   Chain7Long.Drive.ACT.CMD.HwPosOvertravel_Dis := FALSE;
   Chain7Long.Drive.ACT.CMD.HwNegOvertravel_Dis := FALSE;
   Chain7Long.Drive.ACT.CMD.HwOvertravel_MSG_En := FALSE;
   Chain7Long.Drive.ACT.CMD.OneShootMove := FALSE;
   Chain7Long.Drive.ACT.CMD.Move_Type := 3;
   Chain7Long.Drive.ACT.CMD.Target_Pos := 0.0;
   Chain7Long.Drive.ACT.CMD.Speed := 50.0;
   Chain7Long.Drive.ACT.CMD.Acceleration := 300.0;
   Chain7Long.Drive.ACT.CMD.Deceleration := 300.0;
   Chain7Long.Drive.ACT.CMD.Torque_Limit := 30.0;
   Chain7Long.Drive.ACT.CMD.Gear_Ratio := 0.0;
   Chain7Long.Drive.ACT.CMD.Mccp_Length := 2;
   Chain7Long.Drive.ACT.CMD.Mccp_StartSlope := 0.0;
   Chain7Long.Drive.ACT.CMD.Mccp_EndSlope := 0.0;
   Chain7Long.Drive.ACT.CMD.Mapc_Direction := 1;
   Chain7Long.Drive.ACT.CMD.Mapc_SlaveScaling := 1.0;
   Chain7Long.Drive.ACT.CMD.Mapc_MasterScaling := 1.0;
   Chain7Long.Drive.ACT.CMD.Mapc_MasterLockPosition := 0.0;
   Chain7Long.Drive.ACT.CMD.Mapc_CamLockPosition := 0.0;
   Chain7Long.Drive.ACT.CMD.Cam[0].leadingValueStart := 0.0;
   Chain7Long.Drive.ACT.CMD.Cam[1].leadingValueStart := 162.0;
   Chain7Long.Drive.ACT.CMD.Cam[2..39].leadingValueStart := 0.0;
   Chain7Long.Drive.ACT.CMD.Cam[0].leadingValueEnd := 162.0;
   Chain7Long.Drive.ACT.CMD.Cam[1].leadingValueEnd := 360.0;
   Chain7Long.Drive.ACT.CMD.Cam[2..39].leadingValueEnd := 0.0;
   Chain7Long.Drive.ACT.CMD.Cam[0].followingValueStart := 0.0;
   Chain7Long.Drive.ACT.CMD.Cam[1].followingValueStart := 406.399993896484;
   Chain7Long.Drive.ACT.CMD.Cam[2..39].followingValueStart := 0.0;
   Chain7Long.Drive.ACT.CMD.Cam[0..1].followingValueEnd := 406.399993896484;
   Chain7Long.Drive.ACT.CMD.Cam[2..39].followingValueEnd := 0.0;
   Chain7Long.Drive.ACT.CMD.Cam[0..39].geoVeloStart := 0.0;
   Chain7Long.Drive.ACT.CMD.Cam[0..39].geoVeloEnd := 0.0;
   Chain7Long.Drive.ACT.CMD.Cam[0..39].geoAccelStart := 0.0;
   Chain7Long.Drive.ACT.CMD.Cam[0..39].geoAccelEnd := 0.0;
   Chain7Long.Drive.ACT.CMD.Cam[0..39].geoJerkStart := 0.0;
   Chain7Long.Drive.ACT.CMD.Cam[0..39].geoJerkEnd := 0.0;
   Chain7Long.Drive.ACT.CMD.Cam[0..39].inflectionPointParameter := 0.5;
   Chain7Long.Drive.ACT.CMD.Cam[0..39].modVeloTrapezoidParameter := 1.0;
   Chain7Long.Drive.ACT.CMD.Cam[0..39].modSineMaxAccelCaStar := 0.0;
   Chain7Long.Drive.ACT.CMD.Cam[0].camProfileType := 5;
   Chain7Long.Drive.ACT.CMD.Cam[1].camProfileType := 2;
   Chain7Long.Drive.ACT.CMD.Cam[2..39].camProfileType := 0;
   Chain7Long.Drive.ACT.FBK.Ready := TRUE;
   Chain7Long.Drive.ACT.FBK.Calibrated := TRUE;
   Chain7Long.Drive.ACT.FBK.Fault := FALSE;
   Chain7Long.Drive.ACT.FBK.ModuleConnFault := FALSE;
   Chain7Long.Drive.ACT.FBK.In_Position := FALSE;
   Chain7Long.Drive.ACT.FBK.Standstill := TRUE;
   Chain7Long.Drive.ACT.FBK.Enabled := FALSE;
   Chain7Long.Drive.ACT.FBK.BusReadyStatus := FALSE;
   Chain7Long.Drive.ACT.FBK.BrakeReleased := FALSE;
   Chain7Long.Drive.ACT.FBK.HwPosOvertravelDisabled := FALSE;
   Chain7Long.Drive.ACT.FBK.HwNegOvertravelDisabled := FALSE;
   Chain7Long.Drive.ACT.FBK.SafeOffStatus := FALSE;
   Chain7Long.Drive.ACT.FBK.MaxTorqueLimit := FALSE;
   Chain7Long.Drive.ACT.FBK.PosMerge_IP := FALSE;
   Chain7Long.Drive.ACT.FBK.PosMerge_PC := FALSE;
   Chain7Long.Drive.ACT.FBK.Gearing_IP := FALSE;
   Chain7Long.Drive.ACT.FBK.Position := 279.363;
   Chain7Long.Drive.ACT.FBK.Speed := 0.0;
   Chain7Long.Drive.ACT.FBK.Torque := 0.0;
   Chain7Long.Drive.ACT.FBK.RegInput1Pos := 0.0;
   Chain7Long.Drive.ACT.FBK.SeqCamErrorCode := 0;
   Chain7Long.Drive.ACT.FBK.SeqCamTargetPosMAM := 0.0;
   Chain7Long.Drive.ACT.FBK.SeqCamStatus.EndSequence := FALSE;
   Chain7Long.Drive.ACT.FBK.SeqCamStatus.EndSuccess := FALSE;
   Chain7Long.Drive.ACT.FBK.SeqCamStatus.EndError := FALSE;
   Chain7Long.Drive.ACT.FBK.SeqCamStatus.CamHook := FALSE;
   Chain7Long.Drive.ACT.FBK.SeqCamStatus.BothMapc_IP := FALSE;
   Chain7Long.Drive.ACT.FBK.SeqCamStatus.SlaveFwd := FALSE;
   Chain7Long.Drive.ACT.FBK.SeqCamStatus.SlaveBwd := FALSE;
   Chain7Long.Drive.ACT.FBK.SeqCamStatus.SlaveUnwind := FALSE;
   Chain7Long.Drive.ACT.FBK.SeqCamStatus.WaitValidByOpe := FALSE;
   Chain7Long.Drive.ACT.FBK.SeqCamStatus.MapcA_IP := FALSE;
   Chain7Long.Drive.ACT.FBK.SeqCamStatus.MapcB_IP := FALSE;
   Chain7Long.Drive.ACT.FBK.SeqCamStatus.MapcC_IP := FALSE;
   Chain7Long.Drive.ACT.FBK.SeqCamStatus.CamOnce_PC := FALSE;
   Chain7Long.Drive.ACT.FBK.SeqCamStatus.MaxDevError := FALSE;
   Chain7Long.Drive.ACT.FBK.SeqCamStatus.PositionCamLockStatus := FALSE;
   Chain7Long.Drive.ACT.FBK.SeqCamStatus.WaitRestart := FALSE;
   Chain7Long.Drive.ACT.FBK.SeqCamStatus.Bit17 := FALSE;
   Chain7Long.Drive.ACT.FBK.SeqCamStatus.Bit18 := FALSE;
   Chain7Long.Drive.ACT.FBK.SeqCamStatus.Bit19 := FALSE;
   Chain7Long.Drive.ACT.FBK.SeqCamStatus.Bit20 := FALSE;
   Chain7Long.Drive.ACT.FBK.SeqCamStatus.Bit21 := FALSE;
   Chain7Long.Drive.ACT.FBK.SeqCamStatus.Bit22 := FALSE;
   Chain7Long.Drive.ACT.FBK.SeqCamStatus.Bit23 := FALSE;
   Chain7Long.Drive.ACT.FBK.SeqCamStatus.Bit24 := FALSE;
   Chain7Long.Drive.ACT.FBK.SeqCamStatus.Bit25 := FALSE;
   Chain7Long.Drive.ACT.FBK.SeqCamStatus.Bit26 := FALSE;
   Chain7Long.Drive.ACT.FBK.SeqCamStatus.Bit27 := FALSE;
   Chain7Long.Drive.ACT.FBK.SeqCamStatus.Bit28 := FALSE;
   Chain7Long.Drive.ACT.FBK.SeqCamStatus.Bit29 := FALSE;
   Chain7Long.Drive.ACT.FBK.SeqCamStatus.Bit30 := FALSE;
   Chain7Long.Drive.ACT.FBK.SeqCamStatus.Bit31 := FALSE;
   Chain7Long.Drive.ACT.FBK.SeqCamStatus.Bit32 := FALSE;
   Chain7Long.Drive.PLS.FinePosOk.LowLimit := 405.4;
   Chain7Long.Drive.PLS.FinePosOk.HighLimit := 1.0;
   Chain7Long.Drive.PLS.FinePosOk.Ok := FALSE;
   Chain7Long.Drive.PLS.KeepPosOk.LowLimit := 404.4;
   Chain7Long.Drive.PLS.KeepPosOk.HighLimit := 2.0;
   Chain7Long.Drive.PLS.KeepPosOk.Ok := FALSE;
   Chain7Long.Drive.PLS.Up.LowLimit := 0.0;
   Chain7Long.Drive.PLS.Up.HighLimit := 0.0;
   Chain7Long.Drive.PLS.Up.Ok := FALSE;
   Chain7Long.Drive.PLS.Intermediate.LowLimit := 0.0;
   Chain7Long.Drive.PLS.Intermediate.HighLimit := 0.0;
   Chain7Long.Drive.PLS.Intermediate.Ok := FALSE;
   Chain7Long.Drive.PLS.Down.LowLimit := 0.0;
   Chain7Long.Drive.PLS.Down.HighLimit := 0.0;
   Chain7Long.Drive.PLS.Down.Ok := FALSE;
   Chain7Long.Drive.PLS.Forward.LowLimit := 0.0;
   Chain7Long.Drive.PLS.Forward.HighLimit := 0.0;
   Chain7Long.Drive.PLS.Forward.Ok := FALSE;
   Chain7Long.Drive.PLS.Backward.LowLimit := 0.0;
   Chain7Long.Drive.PLS.Backward.HighLimit := 0.0;
   Chain7Long.Drive.PLS.Backward.Ok := FALSE;
   Chain7Long.Drive.PLS.Open.LowLimit := 0.0;
   Chain7Long.Drive.PLS.Open.HighLimit := 0.0;
   Chain7Long.Drive.PLS.Open.Ok := FALSE;
   Chain7Long.Drive.PLS.Close.LowLimit := 0.0;
   Chain7Long.Drive.PLS.Close.HighLimit := 0.0;
   Chain7Long.Drive.PLS.Close.Ok := FALSE;
   Chain7Long.Drive.PLS.PreOpen.LowLimit := 0.0;
   Chain7Long.Drive.PLS.PreOpen.HighLimit := 0.0;
   Chain7Long.Drive.PLS.PreOpen.Ok := FALSE;
   Chain7Long.Drive.PLS.Maintenance.LowLimit := 0.0;
   Chain7Long.Drive.PLS.Maintenance.HighLimit := 0.0;
   Chain7Long.Drive.PLS.Maintenance.Ok := FALSE;
   Chain7Long.Drive.PLS.OperatorSide.LowLimit := 0.0;
   Chain7Long.Drive.PLS.OperatorSide.HighLimit := 0.0;
   Chain7Long.Drive.PLS.OperatorSide.Ok := FALSE;
   Chain7Long.Drive.PLS.NotOperatorSide.LowLimit := 0.0;
   Chain7Long.Drive.PLS.NotOperatorSide.HighLimit := 0.0;
   Chain7Long.Drive.PLS.NotOperatorSide.Ok := FALSE;
   Chain7Long.Drive.PLS.OnMould.LowLimit := 0.0;
   Chain7Long.Drive.PLS.OnMould.HighLimit := 0.0;
   Chain7Long.Drive.PLS.OnMould.Ok := FALSE;
   Chain7Long.Drive.PLS.OffMould.LowLimit := 0.0;
   Chain7Long.Drive.PLS.OffMould.HighLimit := 0.0;
   Chain7Long.Drive.PLS.OffMould.Ok := FALSE;
   Chain7Long.Drive.PLS.Pos0.LowLimit := 0.0;
   Chain7Long.Drive.PLS.Pos0.HighLimit := 0.0;
   Chain7Long.Drive.PLS.Pos0.Ok := FALSE;
   Chain7Long.Drive.PLS.Pos1.LowLimit := 0.0;
   Chain7Long.Drive.PLS.Pos1.HighLimit := 0.0;
   Chain7Long.Drive.PLS.Pos1.Ok := FALSE;
   Chain7Long.Drive.PLS.Pos2.LowLimit := 0.0;
   Chain7Long.Drive.PLS.Pos2.HighLimit := 0.0;
   Chain7Long.Drive.PLS.Pos2.Ok := FALSE;
   Chain7Long.Drive.PLS.Pos3.LowLimit := 0.0;
   Chain7Long.Drive.PLS.Pos3.HighLimit := 0.0;
   Chain7Long.Drive.PLS.Pos3.Ok := FALSE;
   Chain7Long.Drive.PLS.Pos4.LowLimit := 0.0;
   Chain7Long.Drive.PLS.Pos4.HighLimit := 0.0;
   Chain7Long.Drive.PLS.Pos4.Ok := FALSE;
   Chain7Long.Drive.PLS.Pos5.LowLimit := 0.0;
   Chain7Long.Drive.PLS.Pos5.HighLimit := 0.0;
   Chain7Long.Drive.PLS.Pos5.Ok := FALSE;
   Chain7Long.Drive.TON_EnableDrive.PT := T#500MS;
   Chain7Long.Drive.TON_EnableDrive.IN := FALSE;
   Chain7Long.Drive.TON_HwOvertravel_Dis.PT := T#0MS;
   Chain7Long.Drive.TON_HwOvertravel_Dis.IN := FALSE;
   Chain7Long.Drive.TON_HwOvertravel_En.PT := T#0MS;
   Chain7Long.Drive.TON_HwOvertravel_En.IN := FALSE;
   Chain7Long.Drive.TON_TimeoutMovement.PT := T#0MS;
   Chain7Long.Drive.TON_TimeoutMovement.IN := FALSE;
   Chain8Cross.AlmOk := TRUE;
   Chain8Cross.StationWorked := TRUE;
   Chain8Cross.CheckObstruction := FALSE;
   Chain8Cross.OutChainObstruction := TRUE;
   Chain8Cross.StrobeWork := FALSE;
   Chain8Cross.StrobeShift := FALSE;
   Chain8Cross.ManualMovement := FALSE;
   Chain8Cross.OkToStop := TRUE;
   Chain8Cross.PosOk := TRUE;
   Chain8Cross.Ons_PosOk := TRUE;
   Chain8Cross.EnaMove := TRUE;
   Chain8Cross.StationEna := TRUE;
   Chain8Cross.ModeLong := FALSE;
   Chain8Cross.ModeCross := TRUE;
   Chain8Cross.ModeCont := FALSE;
   Chain8Cross.Cfg_Mould_ChainSteps := 1;
   Chain8Cross.Cfg_Mould_EndPos := 8;
   Chain8Cross.Shift_Lenght := 9;
   Chain8Cross.PosMasterAdvanceStep := 0.0;
   Chain8Cross.Input.EndChaMouPre := FALSE;
   Chain8Cross.Input.PshHig := FALSE;
   Chain8Cross.Input.PshLow := FALSE;
   Chain8Cross.Output.PshHig := FALSE;
   Chain8Cross.Output.PshLow := FALSE;
   Chain8Cross.Man.EnaPbt := FALSE;
   Chain8Cross.Man.RstCmd := TRUE;
   Chain8Cross.Man.ScreenNumber := 300_080_301;
   Chain8Cross.Man.WithinScreenRange := 0;
   Chain8Cross.Drive.AlmOk := FALSE;
   Chain8Cross.Drive.AlmEmerg := FALSE;
   Chain8Cross.Drive.AlmNode := FALSE;
   Chain8Cross.Drive.InitPosDrive := FALSE;
   Chain8Cross.Drive.InitPosDrivePLS := FALSE;
   Chain8Cross.Drive.GearingON := FALSE;
   Chain8Cross.Drive.CamHook := FALSE;
   Chain8Cross.Drive.CamStoppingPhase := FALSE;
   Chain8Cross.Drive.RepositioningRequest := FALSE;
   Chain8Cross.Drive.CamRequestResult := FALSE;
   Chain8Cross.Drive.CamRequestError := FALSE;
   Chain8Cross.Drive.CamRequestOk := TRUE;
   Chain8Cross.Drive.CalibDisAxisReq := FALSE;
   Chain8Cross.Drive.CalibReq := FALSE;
   Chain8Cross.Drive.CalibProcess := FALSE;
   Chain8Cross.Drive.HwOvertravelDisReq := FALSE;
   Chain8Cross.Drive.HwOvertravelEnReq := FALSE;
   Chain8Cross.Drive.AuxCamRequest := FALSE;
   Chain8Cross.Drive.TorquePeakEna := TRUE;
   Chain8Cross.Drive.Cmd_Repos := FALSE;
   Chain8Cross.Drive.Ons_CamRequest := FALSE;
   Chain8Cross.Drive.AuxCmdPosition := 0;
   Chain8Cross.Drive.Unwind := 711.2;
   Chain8Cross.Drive.MaxDev := 150.0;
   Chain8Cross.Drive.ReposSpeed := 10.0;
   Chain8Cross.Drive.CalcSlaveDifferenceABS := 0.0;
   Chain8Cross.Drive.CalcModPosition := 0.0;
   Chain8Cross.Drive.CalcSlaveDifference := 0.0;
   Chain8Cross.Drive.CalcMinDeltaPos := 0.0;
   Chain8Cross.Drive.CalcMaxDeltaPos := 0.0;
   Chain8Cross.Drive.CalcHalfPosUnwind := 0.0;
   Chain8Cross.Drive.Man.Cmd_PosJog := FALSE;
   Chain8Cross.Drive.Man.Cmd_NegJog := FALSE;
   Chain8Cross.Drive.Man.Cmd_Step := FALSE;
   Chain8Cross.Drive.Man.Cmd_Forward := FALSE;
   Chain8Cross.Drive.Man.Cmd_Backward := FALSE;
   Chain8Cross.Drive.Man.Cmd_Up := FALSE;
   Chain8Cross.Drive.Man.Cmd_Down := FALSE;
   Chain8Cross.Drive.Man.Cmd_Intermediate := FALSE;
   Chain8Cross.Drive.Man.Cmd_Open := FALSE;
   Chain8Cross.Drive.Man.Cmd_Close := FALSE;
   Chain8Cross.Drive.Man.Cmd_PreOpen := FALSE;
   Chain8Cross.Drive.Man.Cmd_Maintenance := FALSE;
   Chain8Cross.Drive.Man.Cmd_OperatorSide := FALSE;
   Chain8Cross.Drive.Man.Cmd_NotOperatorSide := FALSE;
   Chain8Cross.Drive.Man.Cmd_OnMould := FALSE;
   Chain8Cross.Drive.Man.Cmd_OffMould := FALSE;
   Chain8Cross.Drive.Man.Cmd_Pos0 := FALSE;
   Chain8Cross.Drive.Man.Cmd_Pos1 := FALSE;
   Chain8Cross.Drive.Man.Cmd_Pos2 := FALSE;
   Chain8Cross.Drive.Man.Cmd_Pos3 := FALSE;
   Chain8Cross.Drive.Man.Cmd_Pos4 := FALSE;
   Chain8Cross.Drive.Man.Cmd_Pos5 := FALSE;
   Chain8Cross.Drive.Man.Ons_Step := FALSE;
   Chain8Cross.Drive.Man.PhaseJogCmd := TRUE;
   Chain8Cross.Drive.Man.CmdStartStep := FALSE;
   Chain8Cross.Drive.Man.CmdEndStep := FALSE;
   Chain8Cross.Drive.Man.StepCond := FALSE;
   Chain8Cross.Drive.Man.TON_DelayHomeCmd.PT := T#3S;
   Chain8Cross.Drive.Man.TON_DelayHomeCmd.IN := FALSE;
   Chain8Cross.Drive.Auto.Cmd_Step := FALSE;
   Chain8Cross.Drive.Auto.Cmd_StartStep := FALSE;
   Chain8Cross.Drive.Auto.Cmd_EndStep := FALSE;
   Chain8Cross.Drive.Auto.Cmd_Forward := FALSE;
   Chain8Cross.Drive.Auto.Cmd_Backward := FALSE;
   Chain8Cross.Drive.Auto.Cmd_Up := FALSE;
   Chain8Cross.Drive.Auto.Cmd_Down := FALSE;
   Chain8Cross.Drive.Auto.Cmd_Intermediate := FALSE;
   Chain8Cross.Drive.Auto.Cmd_Open := FALSE;
   Chain8Cross.Drive.Auto.Cmd_Close := FALSE;
   Chain8Cross.Drive.Auto.Cmd_PreOpen := FALSE;
   Chain8Cross.Drive.Auto.Cmd_Maintenance := FALSE;
   Chain8Cross.Drive.Auto.Cmd_OperatorSide := FALSE;
   Chain8Cross.Drive.Auto.Cmd_NotOperatorSide := FALSE;
   Chain8Cross.Drive.Auto.Cmd_OnMould := FALSE;
   Chain8Cross.Drive.Auto.Cmd_OffMould := FALSE;
   Chain8Cross.Drive.Auto.Cmd_Pos0 := FALSE;
   Chain8Cross.Drive.Auto.Cmd_Pos1 := FALSE;
   Chain8Cross.Drive.Auto.Cmd_Pos2 := FALSE;
   Chain8Cross.Drive.Auto.Cmd_Pos3 := FALSE;
   Chain8Cross.Drive.Auto.Cmd_Pos4 := FALSE;
   Chain8Cross.Drive.Auto.Cmd_Pos5 := FALSE;
   Chain8Cross.Drive.Auto.Cmd_Gear := FALSE;
   Chain8Cross.Drive.ACT.CMD.Enable := FALSE;
   Chain8Cross.Drive.ACT.CMD.Pos_Mode := FALSE;
   Chain8Cross.Drive.ACT.CMD.MergeDisabled := FALSE;
   Chain8Cross.Drive.ACT.CMD.SCurve := FALSE;
   Chain8Cross.Drive.ACT.CMD.Cam_Mode := TRUE;
   Chain8Cross.Drive.ACT.CMD.Cam_Request := FALSE;
   Chain8Cross.Drive.ACT.CMD.Cam_PhaseStop := FALSE;
   Chain8Cross.Drive.ACT.CMD.Gear_Mode := FALSE;
   Chain8Cross.Drive.ACT.CMD.Repos_Req := FALSE;
   Chain8Cross.Drive.ACT.CMD.Jog_Pos := FALSE;
   Chain8Cross.Drive.ACT.CMD.Jog_Neg := FALSE;
   Chain8Cross.Drive.ACT.CMD.Stop := FALSE;
   Chain8Cross.Drive.ACT.CMD.Calibration_Req := FALSE;
   Chain8Cross.Drive.ACT.CMD.Reset := FALSE;
   Chain8Cross.Drive.ACT.CMD.RegInput1 := FALSE;
   Chain8Cross.Drive.ACT.CMD.Brake_Release := FALSE;
   Chain8Cross.Drive.ACT.CMD.HwPosOvertravel_Dis := FALSE;
   Chain8Cross.Drive.ACT.CMD.HwNegOvertravel_Dis := FALSE;
   Chain8Cross.Drive.ACT.CMD.HwOvertravel_MSG_En := FALSE;
   Chain8Cross.Drive.ACT.CMD.OneShootMove := FALSE;
   Chain8Cross.Drive.ACT.CMD.Move_Type := 3;
   Chain8Cross.Drive.ACT.CMD.Target_Pos := 0.0;
   Chain8Cross.Drive.ACT.CMD.Speed := 0.0;
   Chain8Cross.Drive.ACT.CMD.Acceleration := 300.0;
   Chain8Cross.Drive.ACT.CMD.Deceleration := 300.0;
   Chain8Cross.Drive.ACT.CMD.Torque_Limit := 30.0;
   Chain8Cross.Drive.ACT.CMD.Gear_Ratio := 0.0;
   Chain8Cross.Drive.ACT.CMD.Mccp_Length := 6;
   Chain8Cross.Drive.ACT.CMD.Mccp_StartSlope := 0.0;
   Chain8Cross.Drive.ACT.CMD.Mccp_EndSlope := 0.0;
   Chain8Cross.Drive.ACT.CMD.Mapc_Direction := 1;
   Chain8Cross.Drive.ACT.CMD.Mapc_SlaveScaling := 1.0;
   Chain8Cross.Drive.ACT.CMD.Mapc_MasterScaling := 1.0;
   Chain8Cross.Drive.ACT.CMD.Mapc_MasterLockPosition := 0.0;
   Chain8Cross.Drive.ACT.CMD.Mapc_CamLockPosition := 0.0;
   Chain8Cross.Drive.ACT.CMD.Cam[0].leadingValueStart := 0.0;
   Chain8Cross.Drive.ACT.CMD.Cam[1].leadingValueStart := 193.679992675781;
   Chain8Cross.Drive.ACT.CMD.Cam[2..3].leadingValueStart := 225.360000610352;
   Chain8Cross.Drive.ACT.CMD.Cam[4].leadingValueStart := 328.320007324219;
   Chain8Cross.Drive.ACT.CMD.Cam[5].leadingValueStart := 360.0;
   Chain8Cross.Drive.ACT.CMD.Cam[6..39].leadingValueStart := 0.0;
   Chain8Cross.Drive.ACT.CMD.Cam[0].leadingValueEnd := 162.0;
   Chain8Cross.Drive.ACT.CMD.Cam[1..2].leadingValueEnd := 0.0;
   Chain8Cross.Drive.ACT.CMD.Cam[3].leadingValueEnd := 296.640014648438;
   Chain8Cross.Drive.ACT.CMD.Cam[4..39].leadingValueEnd := 0.0;
   Chain8Cross.Drive.ACT.CMD.Cam[0].followingValueStart := 0.0;
   Chain8Cross.Drive.ACT.CMD.Cam[1].followingValueStart := 27.8901958465576;
   Chain8Cross.Drive.ACT.CMD.Cam[2..3].followingValueStart := 167.341171264648;
   Chain8Cross.Drive.ACT.CMD.Cam[4].followingValueStart := 683.309753417969;
   Chain8Cross.Drive.ACT.CMD.Cam[5].followingValueStart := 711.200012207031;
   Chain8Cross.Drive.ACT.CMD.Cam[6..39].followingValueStart := 0.0;
   Chain8Cross.Drive.ACT.CMD.Cam[0..2].followingValueEnd := 0.0;
   Chain8Cross.Drive.ACT.CMD.Cam[3].followingValueEnd := 543.858825683594;
   Chain8Cross.Drive.ACT.CMD.Cam[4..39].followingValueEnd := 0.0;
   Chain8Cross.Drive.ACT.CMD.Cam[0..39].geoVeloStart := 0.0;
   Chain8Cross.Drive.ACT.CMD.Cam[0..39].geoVeloEnd := 0.0;
   Chain8Cross.Drive.ACT.CMD.Cam[0..39].geoAccelStart := 0.0;
   Chain8Cross.Drive.ACT.CMD.Cam[0..39].geoAccelEnd := 0.0;
   Chain8Cross.Drive.ACT.CMD.Cam[0..39].geoJerkStart := 0.0;
   Chain8Cross.Drive.ACT.CMD.Cam[0..39].geoJerkEnd := 0.0;
   Chain8Cross.Drive.ACT.CMD.Cam[0..39].inflectionPointParameter := 0.5;
   Chain8Cross.Drive.ACT.CMD.Cam[0..39].modVeloTrapezoidParameter := 1.0;
   Chain8Cross.Drive.ACT.CMD.Cam[0..39].modSineMaxAccelCaStar := 0.0;
   Chain8Cross.Drive.ACT.CMD.Cam[0].camProfileType := 2;
   Chain8Cross.Drive.ACT.CMD.Cam[1..2].camProfileType := 1;
   Chain8Cross.Drive.ACT.CMD.Cam[3].camProfileType := 3;
   Chain8Cross.Drive.ACT.CMD.Cam[4..5].camProfileType := 1;
   Chain8Cross.Drive.ACT.CMD.Cam[6..39].camProfileType := 0;
   Chain8Cross.Drive.ACT.FBK.Ready := TRUE;
   Chain8Cross.Drive.ACT.FBK.Calibrated := TRUE;
   Chain8Cross.Drive.ACT.FBK.Fault := FALSE;
   Chain8Cross.Drive.ACT.FBK.ModuleConnFault := FALSE;
   Chain8Cross.Drive.ACT.FBK.In_Position := FALSE;
   Chain8Cross.Drive.ACT.FBK.Standstill := TRUE;
   Chain8Cross.Drive.ACT.FBK.Enabled := FALSE;
   Chain8Cross.Drive.ACT.FBK.BusReadyStatus := FALSE;
   Chain8Cross.Drive.ACT.FBK.BrakeReleased := FALSE;
   Chain8Cross.Drive.ACT.FBK.HwPosOvertravelDisabled := FALSE;
   Chain8Cross.Drive.ACT.FBK.HwNegOvertravelDisabled := FALSE;
   Chain8Cross.Drive.ACT.FBK.SafeOffStatus := FALSE;
   Chain8Cross.Drive.ACT.FBK.MaxTorqueLimit := FALSE;
   Chain8Cross.Drive.ACT.FBK.PosMerge_IP := FALSE;
   Chain8Cross.Drive.ACT.FBK.PosMerge_PC := FALSE;
   Chain8Cross.Drive.ACT.FBK.Gearing_IP := FALSE;
   Chain8Cross.Drive.ACT.FBK.Position := 0.078;
   Chain8Cross.Drive.ACT.FBK.Speed := 0.0;
   Chain8Cross.Drive.ACT.FBK.Torque := 0.0;
   Chain8Cross.Drive.ACT.FBK.RegInput1Pos := 0.0;
   Chain8Cross.Drive.ACT.FBK.SeqCamErrorCode := 0;
   Chain8Cross.Drive.ACT.FBK.SeqCamTargetPosMAM := 0.0;
   Chain8Cross.Drive.ACT.FBK.SeqCamStatus.EndSequence := FALSE;
   Chain8Cross.Drive.ACT.FBK.SeqCamStatus.EndSuccess := FALSE;
   Chain8Cross.Drive.ACT.FBK.SeqCamStatus.EndError := FALSE;
   Chain8Cross.Drive.ACT.FBK.SeqCamStatus.CamHook := FALSE;
   Chain8Cross.Drive.ACT.FBK.SeqCamStatus.BothMapc_IP := FALSE;
   Chain8Cross.Drive.ACT.FBK.SeqCamStatus.SlaveFwd := FALSE;
   Chain8Cross.Drive.ACT.FBK.SeqCamStatus.SlaveBwd := FALSE;
   Chain8Cross.Drive.ACT.FBK.SeqCamStatus.SlaveUnwind := FALSE;
   Chain8Cross.Drive.ACT.FBK.SeqCamStatus.WaitValidByOpe := FALSE;
   Chain8Cross.Drive.ACT.FBK.SeqCamStatus.MapcA_IP := FALSE;
   Chain8Cross.Drive.ACT.FBK.SeqCamStatus.MapcB_IP := FALSE;
   Chain8Cross.Drive.ACT.FBK.SeqCamStatus.MapcC_IP := FALSE;
   Chain8Cross.Drive.ACT.FBK.SeqCamStatus.CamOnce_PC := FALSE;
   Chain8Cross.Drive.ACT.FBK.SeqCamStatus.MaxDevError := FALSE;
   Chain8Cross.Drive.ACT.FBK.SeqCamStatus.PositionCamLockStatus := FALSE;
   Chain8Cross.Drive.ACT.FBK.SeqCamStatus.WaitRestart := FALSE;
   Chain8Cross.Drive.ACT.FBK.SeqCamStatus.Bit17 := FALSE;
   Chain8Cross.Drive.ACT.FBK.SeqCamStatus.Bit18 := FALSE;
   Chain8Cross.Drive.ACT.FBK.SeqCamStatus.Bit19 := FALSE;
   Chain8Cross.Drive.ACT.FBK.SeqCamStatus.Bit20 := FALSE;
   Chain8Cross.Drive.ACT.FBK.SeqCamStatus.Bit21 := FALSE;
   Chain8Cross.Drive.ACT.FBK.SeqCamStatus.Bit22 := FALSE;
   Chain8Cross.Drive.ACT.FBK.SeqCamStatus.Bit23 := FALSE;
   Chain8Cross.Drive.ACT.FBK.SeqCamStatus.Bit24 := FALSE;
   Chain8Cross.Drive.ACT.FBK.SeqCamStatus.Bit25 := FALSE;
   Chain8Cross.Drive.ACT.FBK.SeqCamStatus.Bit26 := FALSE;
   Chain8Cross.Drive.ACT.FBK.SeqCamStatus.Bit27 := FALSE;
   Chain8Cross.Drive.ACT.FBK.SeqCamStatus.Bit28 := FALSE;
   Chain8Cross.Drive.ACT.FBK.SeqCamStatus.Bit29 := FALSE;
   Chain8Cross.Drive.ACT.FBK.SeqCamStatus.Bit30 := FALSE;
   Chain8Cross.Drive.ACT.FBK.SeqCamStatus.Bit31 := FALSE;
   Chain8Cross.Drive.ACT.FBK.SeqCamStatus.Bit32 := FALSE;
   Chain8Cross.Drive.PLS.FinePosOk.LowLimit := 710.2;
   Chain8Cross.Drive.PLS.FinePosOk.HighLimit := 1.0;
   Chain8Cross.Drive.PLS.FinePosOk.Ok := TRUE;
   Chain8Cross.Drive.PLS.KeepPosOk.LowLimit := 709.2;
   Chain8Cross.Drive.PLS.KeepPosOk.HighLimit := 2.0;
   Chain8Cross.Drive.PLS.KeepPosOk.Ok := TRUE;
   Chain8Cross.Drive.PLS.Up.LowLimit := 0.0;
   Chain8Cross.Drive.PLS.Up.HighLimit := 0.0;
   Chain8Cross.Drive.PLS.Up.Ok := FALSE;
   Chain8Cross.Drive.PLS.Intermediate.LowLimit := 0.0;
   Chain8Cross.Drive.PLS.Intermediate.HighLimit := 0.0;
   Chain8Cross.Drive.PLS.Intermediate.Ok := FALSE;
   Chain8Cross.Drive.PLS.Down.LowLimit := 0.0;
   Chain8Cross.Drive.PLS.Down.HighLimit := 0.0;
   Chain8Cross.Drive.PLS.Down.Ok := FALSE;
   Chain8Cross.Drive.PLS.Forward.LowLimit := 0.0;
   Chain8Cross.Drive.PLS.Forward.HighLimit := 0.0;
   Chain8Cross.Drive.PLS.Forward.Ok := FALSE;
   Chain8Cross.Drive.PLS.Backward.LowLimit := 0.0;
   Chain8Cross.Drive.PLS.Backward.HighLimit := 0.0;
   Chain8Cross.Drive.PLS.Backward.Ok := FALSE;
   Chain8Cross.Drive.PLS.Open.LowLimit := 0.0;
   Chain8Cross.Drive.PLS.Open.HighLimit := 0.0;
   Chain8Cross.Drive.PLS.Open.Ok := FALSE;
   Chain8Cross.Drive.PLS.Close.LowLimit := 0.0;
   Chain8Cross.Drive.PLS.Close.HighLimit := 0.0;
   Chain8Cross.Drive.PLS.Close.Ok := FALSE;
   Chain8Cross.Drive.PLS.PreOpen.LowLimit := 0.0;
   Chain8Cross.Drive.PLS.PreOpen.HighLimit := 0.0;
   Chain8Cross.Drive.PLS.PreOpen.Ok := FALSE;
   Chain8Cross.Drive.PLS.Maintenance.LowLimit := 0.0;
   Chain8Cross.Drive.PLS.Maintenance.HighLimit := 0.0;
   Chain8Cross.Drive.PLS.Maintenance.Ok := FALSE;
   Chain8Cross.Drive.PLS.OperatorSide.LowLimit := 0.0;
   Chain8Cross.Drive.PLS.OperatorSide.HighLimit := 0.0;
   Chain8Cross.Drive.PLS.OperatorSide.Ok := FALSE;
   Chain8Cross.Drive.PLS.NotOperatorSide.LowLimit := 0.0;
   Chain8Cross.Drive.PLS.NotOperatorSide.HighLimit := 0.0;
   Chain8Cross.Drive.PLS.NotOperatorSide.Ok := FALSE;
   Chain8Cross.Drive.PLS.OnMould.LowLimit := 0.0;
   Chain8Cross.Drive.PLS.OnMould.HighLimit := 0.0;
   Chain8Cross.Drive.PLS.OnMould.Ok := FALSE;
   Chain8Cross.Drive.PLS.OffMould.LowLimit := 0.0;
   Chain8Cross.Drive.PLS.OffMould.HighLimit := 0.0;
   Chain8Cross.Drive.PLS.OffMould.Ok := FALSE;
   Chain8Cross.Drive.PLS.Pos0.LowLimit := 0.0;
   Chain8Cross.Drive.PLS.Pos0.HighLimit := 0.0;
   Chain8Cross.Drive.PLS.Pos0.Ok := FALSE;
   Chain8Cross.Drive.PLS.Pos1.LowLimit := 0.0;
   Chain8Cross.Drive.PLS.Pos1.HighLimit := 0.0;
   Chain8Cross.Drive.PLS.Pos1.Ok := FALSE;
   Chain8Cross.Drive.PLS.Pos2.LowLimit := 0.0;
   Chain8Cross.Drive.PLS.Pos2.HighLimit := 0.0;
   Chain8Cross.Drive.PLS.Pos2.Ok := FALSE;
   Chain8Cross.Drive.PLS.Pos3.LowLimit := 0.0;
   Chain8Cross.Drive.PLS.Pos3.HighLimit := 0.0;
   Chain8Cross.Drive.PLS.Pos3.Ok := FALSE;
   Chain8Cross.Drive.PLS.Pos4.LowLimit := 0.0;
   Chain8Cross.Drive.PLS.Pos4.HighLimit := 0.0;
   Chain8Cross.Drive.PLS.Pos4.Ok := FALSE;
   Chain8Cross.Drive.PLS.Pos5.LowLimit := 0.0;
   Chain8Cross.Drive.PLS.Pos5.HighLimit := 0.0;
   Chain8Cross.Drive.PLS.Pos5.Ok := FALSE;
   Chain8Cross.Drive.TON_EnableDrive.PT := T#500MS;
   Chain8Cross.Drive.TON_EnableDrive.IN := FALSE;
   Chain8Cross.Drive.TON_HwOvertravel_Dis.PT := T#0MS;
   Chain8Cross.Drive.TON_HwOvertravel_Dis.IN := FALSE;
   Chain8Cross.Drive.TON_HwOvertravel_En.PT := T#0MS;
   Chain8Cross.Drive.TON_HwOvertravel_En.IN := FALSE;
   Chain8Cross.Drive.TON_TimeoutMovement.PT := T#0MS;
   Chain8Cross.Drive.TON_TimeoutMovement.IN := FALSE;
   VMaster.AtSpeed := TRUE;
   VMaster.AuxStartLongChain := FALSE;
   VMaster.AuxStartCrossChain := FALSE;
   VMaster.Speed_DegSec := 150.0;
   VMaster.PosLongStep := 162.0;
   VMaster.PosCrossStart := 162.0;
   VMaster.PosAscentColumnStart := 0.0;
   VMaster.PosTransferEnd := 192.0;
   VMaster.PosLongChainStepEnd := 162.0;
   VMaster.PosAdvanceCheck := 60.0;
   VMaster.PosAdvanceLongStep := 0.0;
   VMaster.PosAdvanceCrossStep := 0.0;
   VMaster.PosMacStepToStepEnd := 212.0;
   VMaster.Man.EnaPbt := FALSE;
   VMaster.Man.RstCmd := FALSE;
   VMaster.Man.ScreenNumber := 300_090_301;
   VMaster.Man.WithinScreenRange := 0;
   VMaster.Virtual.AlmOk := TRUE;
   VMaster.Virtual.AlmEmerg := FALSE;
   VMaster.Virtual.AlmNode := FALSE;
   VMaster.Virtual.InitPosDrive := FALSE;
   VMaster.Virtual.InitPosDrivePLS := FALSE;
   VMaster.Virtual.GearingON := FALSE;
   VMaster.Virtual.CamHook := FALSE;
   VMaster.Virtual.CamStoppingPhase := FALSE;
   VMaster.Virtual.RepositioningRequest := FALSE;
   VMaster.Virtual.CamRequestResult := FALSE;
   VMaster.Virtual.CamRequestError := FALSE;
   VMaster.Virtual.CamRequestOk := FALSE;
   VMaster.Virtual.AuxCamRequest := FALSE;
   VMaster.Virtual.Cmd_Repos := FALSE;
   VMaster.Virtual.Ons_RedefinePosition := FALSE;
   VMaster.Virtual.Ons_CamRequest := FALSE;
   VMaster.Virtual.AuxCmdPosition := 0;
   VMaster.Virtual.Cfg_FBK_In_Position_Delay_ms := 100;
   VMaster.Virtual.Unwind := 360.0;
   VMaster.Virtual.MaxDev := 0.0;
   VMaster.Virtual.ReposSpeed := 0.0;
   VMaster.Virtual.CalcSlaveDifferenceABS := 0.0;
   VMaster.Virtual.CalcModPosition := 0.0;
   VMaster.Virtual.CalcSlaveDifference := 0.0;
   VMaster.Virtual.CalcMinDeltaPos := 0.0;
   VMaster.Virtual.CalcMaxDeltaPos := 0.0;
   VMaster.Virtual.CalcHalfPosUnwind := 0.0;
   VMaster.Virtual.Man.Cmd_PosJog := FALSE;
   VMaster.Virtual.Man.Cmd_NegJog := FALSE;
   VMaster.Virtual.Man.Cmd_Step := FALSE;
   VMaster.Virtual.Man.Cmd_Forward := FALSE;
   VMaster.Virtual.Man.Cmd_Backward := FALSE;
   VMaster.Virtual.Man.Cmd_Up := FALSE;
   VMaster.Virtual.Man.Cmd_Down := FALSE;
   VMaster.Virtual.Man.Cmd_Intermediate := FALSE;
   VMaster.Virtual.Man.Cmd_Open := FALSE;
   VMaster.Virtual.Man.Cmd_Close := FALSE;
   VMaster.Virtual.Man.Cmd_PreOpen := FALSE;
   VMaster.Virtual.Man.Cmd_Maintenance := FALSE;
   VMaster.Virtual.Man.Cmd_OperatorSide := FALSE;
   VMaster.Virtual.Man.Cmd_NotOperatorSide := FALSE;
   VMaster.Virtual.Man.Cmd_OnMould := FALSE;
   VMaster.Virtual.Man.Cmd_OffMould := FALSE;
   VMaster.Virtual.Man.Cmd_Pos0 := FALSE;
   VMaster.Virtual.Man.Cmd_Pos1 := FALSE;
   VMaster.Virtual.Man.Cmd_Pos2 := FALSE;
   VMaster.Virtual.Man.Cmd_Pos3 := FALSE;
   VMaster.Virtual.Man.Cmd_Pos4 := FALSE;
   VMaster.Virtual.Man.Cmd_Pos5 := FALSE;
   VMaster.Virtual.Man.Ons_Step := FALSE;
   VMaster.Virtual.Man.PhaseJogCmd := FALSE;
   VMaster.Virtual.Man.CmdStartStep := FALSE;
   VMaster.Virtual.Man.CmdEndStep := FALSE;
   VMaster.Virtual.Man.StepCond := FALSE;
   VMaster.Virtual.Man.TON_DelayHomeCmd.PT := T#3S;
   VMaster.Virtual.Man.TON_DelayHomeCmd.IN := FALSE;
   VMaster.Virtual.Auto.Cmd_Step := FALSE;
   VMaster.Virtual.Auto.Cmd_StartStep := FALSE;
   VMaster.Virtual.Auto.Cmd_EndStep := FALSE;
   VMaster.Virtual.Auto.Cmd_Forward := FALSE;
   VMaster.Virtual.Auto.Cmd_Backward := FALSE;
   VMaster.Virtual.Auto.Cmd_Up := FALSE;
   VMaster.Virtual.Auto.Cmd_Down := FALSE;
   VMaster.Virtual.Auto.Cmd_Intermediate := FALSE;
   VMaster.Virtual.Auto.Cmd_Open := FALSE;
   VMaster.Virtual.Auto.Cmd_Close := FALSE;
   VMaster.Virtual.Auto.Cmd_PreOpen := FALSE;
   VMaster.Virtual.Auto.Cmd_Maintenance := FALSE;
   VMaster.Virtual.Auto.Cmd_OperatorSide := FALSE;
   VMaster.Virtual.Auto.Cmd_NotOperatorSide := FALSE;
   VMaster.Virtual.Auto.Cmd_OnMould := FALSE;
   VMaster.Virtual.Auto.Cmd_OffMould := FALSE;
   VMaster.Virtual.Auto.Cmd_Pos0 := FALSE;
   VMaster.Virtual.Auto.Cmd_Pos1 := FALSE;
   VMaster.Virtual.Auto.Cmd_Pos2 := FALSE;
   VMaster.Virtual.Auto.Cmd_Pos3 := FALSE;
   VMaster.Virtual.Auto.Cmd_Pos4 := FALSE;
   VMaster.Virtual.Auto.Cmd_Pos5 := FALSE;
   VMaster.Virtual.Auto.Cmd_Gear := FALSE;
   VMaster.Virtual.ACT.CMD.Enable := TRUE;
   VMaster.Virtual.ACT.CMD.Pos_Mode := FALSE;
   VMaster.Virtual.ACT.CMD.MergeDisabled := FALSE;
   VMaster.Virtual.ACT.CMD.SCurve := FALSE;
   VMaster.Virtual.ACT.CMD.Cam_Mode := FALSE;
   VMaster.Virtual.ACT.CMD.Cam_Request := FALSE;
   VMaster.Virtual.ACT.CMD.Cam_PhaseStop := FALSE;
   VMaster.Virtual.ACT.CMD.Gear_Mode := FALSE;
   VMaster.Virtual.ACT.CMD.Repos_Req := FALSE;
   VMaster.Virtual.ACT.CMD.Jog_Pos := FALSE;
   VMaster.Virtual.ACT.CMD.Jog_Neg := FALSE;
   VMaster.Virtual.ACT.CMD.Stop := TRUE;
   VMaster.Virtual.ACT.CMD.Stop_InPhase := FALSE;
   VMaster.Virtual.ACT.CMD.Stop_Emergency := FALSE;
   VMaster.Virtual.ACT.CMD.Stop_Immediate := FALSE;
   VMaster.Virtual.ACT.CMD.RedefinePosition := FALSE;
   VMaster.Virtual.ACT.CMD.Calibration_Req := FALSE;
   VMaster.Virtual.ACT.CMD.Reset := FALSE;
   VMaster.Virtual.ACT.CMD.OneShootMove := FALSE;
   VMaster.Virtual.ACT.CMD.SetPositionUnwind := FALSE;
   VMaster.Virtual.ACT.CMD.Move_Type := 3;
   VMaster.Virtual.ACT.CMD.Target_Pos := 162.0;
   VMaster.Virtual.ACT.CMD.Speed := 60.0;
   VMaster.Virtual.ACT.CMD.Acceleration := 500.0;
   VMaster.Virtual.ACT.CMD.Deceleration := 750.0;
   VMaster.Virtual.ACT.CMD.PositionUnwind := 0;
   VMaster.Virtual.ACT.CMD.Mrp_Position := 0.0;
   VMaster.Virtual.ACT.CMD.Gear_Ratio := 0.0;
   VMaster.Virtual.ACT.CMD.Mccp_Length := 0;
   VMaster.Virtual.ACT.CMD.Mccp_StartSlope := 0.0;
   VMaster.Virtual.ACT.CMD.Mccp_EndSlope := 0.0;
   VMaster.Virtual.ACT.CMD.Mapc_Direction := 0;
   VMaster.Virtual.ACT.CMD.Mapc_SlaveScaling := 0.0;
   VMaster.Virtual.ACT.CMD.Mapc_MasterScaling := 0.0;
   VMaster.Virtual.ACT.CMD.Mapc_MasterLockPosition := 0.0;
   VMaster.Virtual.ACT.CMD.Mapc_CamLockPosition := 0.0;
   VMaster.Virtual.ACT.CMD.Cam[0..39].leadingValueStart := 0.0;
   VMaster.Virtual.ACT.CMD.Cam[0..39].leadingValueEnd := 0.0;
   VMaster.Virtual.ACT.CMD.Cam[0..39].followingValueStart := 0.0;
   VMaster.Virtual.ACT.CMD.Cam[0..39].followingValueEnd := 0.0;
   VMaster.Virtual.ACT.CMD.Cam[0..39].geoVeloStart := 0.0;
   VMaster.Virtual.ACT.CMD.Cam[0..39].geoVeloEnd := 0.0;
   VMaster.Virtual.ACT.CMD.Cam[0..39].geoAccelStart := 0.0;
   VMaster.Virtual.ACT.CMD.Cam[0..39].geoAccelEnd := 0.0;
   VMaster.Virtual.ACT.CMD.Cam[0..39].geoJerkStart := 0.0;
   VMaster.Virtual.ACT.CMD.Cam[0..39].geoJerkEnd := 0.0;
   VMaster.Virtual.ACT.CMD.Cam[0..39].inflectionPointParameter := 0.5;
   VMaster.Virtual.ACT.CMD.Cam[0..39].modVeloTrapezoidParameter := 1.0;
   VMaster.Virtual.ACT.CMD.Cam[0..39].modSineMaxAccelCaStar := 0.0;
   VMaster.Virtual.ACT.CMD.Cam[0..39].camProfileType := 0;
   VMaster.Virtual.ACT.FBK.Ready := TRUE;
   VMaster.Virtual.ACT.FBK.Calibrated := TRUE;
   VMaster.Virtual.ACT.FBK.MRP_DN := FALSE;
   VMaster.Virtual.ACT.FBK.Fault := FALSE;
   VMaster.Virtual.ACT.FBK.In_Position := TRUE;
   VMaster.Virtual.ACT.FBK.Standstill := TRUE;
   VMaster.Virtual.ACT.FBK.Enabled := TRUE;
   VMaster.Virtual.ACT.FBK.Gearing_IP := FALSE;
   VMaster.Virtual.ACT.FBK.Position := 97.68;
   VMaster.Virtual.ACT.FBK.Speed := 0.0;
   VMaster.Virtual.ACT.FBK.PositionUnwind := 0;
   VMaster.Virtual.ACT.FBK.SeqCamErrorCode := 0;
   VMaster.Virtual.ACT.FBK.SeqCamTargetPosMAM := 0.0;
   VMaster.Virtual.ACT.FBK.SeqCamStatus.EndSequence := FALSE;
   VMaster.Virtual.ACT.FBK.SeqCamStatus.EndSuccess := FALSE;
   VMaster.Virtual.ACT.FBK.SeqCamStatus.EndError := FALSE;
   VMaster.Virtual.ACT.FBK.SeqCamStatus.CamHook := FALSE;
   VMaster.Virtual.ACT.FBK.SeqCamStatus.BothMapc_IP := FALSE;
   VMaster.Virtual.ACT.FBK.SeqCamStatus.SlaveFwd := FALSE;
   VMaster.Virtual.ACT.FBK.SeqCamStatus.SlaveBwd := FALSE;
   VMaster.Virtual.ACT.FBK.SeqCamStatus.SlaveUnwind := FALSE;
   VMaster.Virtual.ACT.FBK.SeqCamStatus.WaitValidByOpe := FALSE;
   VMaster.Virtual.ACT.FBK.SeqCamStatus.MapcA_IP := FALSE;
   VMaster.Virtual.ACT.FBK.SeqCamStatus.MapcB_IP := FALSE;
   VMaster.Virtual.ACT.FBK.SeqCamStatus.MapcC_IP := FALSE;
   VMaster.Virtual.ACT.FBK.SeqCamStatus.CamOnce_PC := FALSE;
   VMaster.Virtual.ACT.FBK.SeqCamStatus.MaxDevError := FALSE;
   VMaster.Virtual.ACT.FBK.SeqCamStatus.PositionCamLockStatus := FALSE;
   VMaster.Virtual.ACT.FBK.SeqCamStatus.WaitRestart := FALSE;
   VMaster.Virtual.ACT.FBK.SeqCamStatus.Bit17 := FALSE;
   VMaster.Virtual.ACT.FBK.SeqCamStatus.Bit18 := FALSE;
   VMaster.Virtual.ACT.FBK.SeqCamStatus.Bit19 := FALSE;
   VMaster.Virtual.ACT.FBK.SeqCamStatus.Bit20 := FALSE;
   VMaster.Virtual.ACT.FBK.SeqCamStatus.Bit21 := FALSE;
   VMaster.Virtual.ACT.FBK.SeqCamStatus.Bit22 := FALSE;
   VMaster.Virtual.ACT.FBK.SeqCamStatus.Bit23 := FALSE;
   VMaster.Virtual.ACT.FBK.SeqCamStatus.Bit24 := FALSE;
   VMaster.Virtual.ACT.FBK.SeqCamStatus.Bit25 := FALSE;
   VMaster.Virtual.ACT.FBK.SeqCamStatus.Bit26 := FALSE;
   VMaster.Virtual.ACT.FBK.SeqCamStatus.Bit27 := FALSE;
   VMaster.Virtual.ACT.FBK.SeqCamStatus.Bit28 := FALSE;
   VMaster.Virtual.ACT.FBK.SeqCamStatus.Bit29 := FALSE;
   VMaster.Virtual.ACT.FBK.SeqCamStatus.Bit30 := FALSE;
   VMaster.Virtual.ACT.FBK.SeqCamStatus.Bit31 := FALSE;
   VMaster.Virtual.ACT.FBK.SeqCamStatus.Bit32 := FALSE;
   VMaster.Virtual.PLS.FinePosOk.LowLimit := 0.0;
   VMaster.Virtual.PLS.FinePosOk.HighLimit := 0.0;
   VMaster.Virtual.PLS.FinePosOk.Ok := FALSE;
   VMaster.Virtual.PLS.KeepPosOk.LowLimit := 0.0;
   VMaster.Virtual.PLS.KeepPosOk.HighLimit := 0.0;
   VMaster.Virtual.PLS.KeepPosOk.Ok := FALSE;
   VMaster.Virtual.PLS.Up.LowLimit := 0.0;
   VMaster.Virtual.PLS.Up.HighLimit := 0.0;
   VMaster.Virtual.PLS.Up.Ok := FALSE;
   VMaster.Virtual.PLS.Intermediate.LowLimit := 0.0;
   VMaster.Virtual.PLS.Intermediate.HighLimit := 0.0;
   VMaster.Virtual.PLS.Intermediate.Ok := FALSE;
   VMaster.Virtual.PLS.Down.LowLimit := 0.0;
   VMaster.Virtual.PLS.Down.HighLimit := 0.0;
   VMaster.Virtual.PLS.Down.Ok := FALSE;
   VMaster.Virtual.PLS.Forward.LowLimit := 0.0;
   VMaster.Virtual.PLS.Forward.HighLimit := 0.0;
   VMaster.Virtual.PLS.Forward.Ok := TRUE;
   VMaster.Virtual.PLS.Backward.LowLimit := 0.0;
   VMaster.Virtual.PLS.Backward.HighLimit := 0.0;
   VMaster.Virtual.PLS.Backward.Ok := FALSE;
   VMaster.Virtual.PLS.Open.LowLimit := 0.0;
   VMaster.Virtual.PLS.Open.HighLimit := 0.0;
   VMaster.Virtual.PLS.Open.Ok := FALSE;
   VMaster.Virtual.PLS.Close.LowLimit := 0.0;
   VMaster.Virtual.PLS.Close.HighLimit := 0.0;
   VMaster.Virtual.PLS.Close.Ok := FALSE;
   VMaster.Virtual.PLS.PreOpen.LowLimit := 0.0;
   VMaster.Virtual.PLS.PreOpen.HighLimit := 0.0;
   VMaster.Virtual.PLS.PreOpen.Ok := FALSE;
   VMaster.Virtual.PLS.Maintenance.LowLimit := 0.0;
   VMaster.Virtual.PLS.Maintenance.HighLimit := 0.0;
   VMaster.Virtual.PLS.Maintenance.Ok := FALSE;
   VMaster.Virtual.PLS.OperatorSide.LowLimit := 0.0;
   VMaster.Virtual.PLS.OperatorSide.HighLimit := 0.0;
   VMaster.Virtual.PLS.OperatorSide.Ok := FALSE;
   VMaster.Virtual.PLS.NotOperatorSide.LowLimit := 0.0;
   VMaster.Virtual.PLS.NotOperatorSide.HighLimit := 0.0;
   VMaster.Virtual.PLS.NotOperatorSide.Ok := FALSE;
   VMaster.Virtual.PLS.OnMould.LowLimit := 0.0;
   VMaster.Virtual.PLS.OnMould.HighLimit := 0.0;
   VMaster.Virtual.PLS.OnMould.Ok := FALSE;
   VMaster.Virtual.PLS.OffMould.LowLimit := 0.0;
   VMaster.Virtual.PLS.OffMould.HighLimit := 0.0;
   VMaster.Virtual.PLS.OffMould.Ok := FALSE;
   VMaster.Virtual.PLS.Pos0.LowLimit := 0.0;
   VMaster.Virtual.PLS.Pos0.HighLimit := 0.0;
   VMaster.Virtual.PLS.Pos0.Ok := FALSE;
   VMaster.Virtual.PLS.Pos1.LowLimit := 0.0;
   VMaster.Virtual.PLS.Pos1.HighLimit := 0.0;
   VMaster.Virtual.PLS.Pos1.Ok := FALSE;
   VMaster.Virtual.PLS.Pos2.LowLimit := 0.0;
   VMaster.Virtual.PLS.Pos2.HighLimit := 0.0;
   VMaster.Virtual.PLS.Pos2.Ok := FALSE;
   VMaster.Virtual.PLS.Pos3.LowLimit := 0.0;
   VMaster.Virtual.PLS.Pos3.HighLimit := 0.0;
   VMaster.Virtual.PLS.Pos3.Ok := FALSE;
   VMaster.Virtual.PLS.Pos4.LowLimit := 0.0;
   VMaster.Virtual.PLS.Pos4.HighLimit := 0.0;
   VMaster.Virtual.PLS.Pos4.Ok := FALSE;
   VMaster.Virtual.PLS.Pos5.LowLimit := 0.0;
   VMaster.Virtual.PLS.Pos5.HighLimit := 0.0;
   VMaster.Virtual.PLS.Pos5.Ok := FALSE;
   VMaster.Virtual.TON_TimeoutMovement.PT := T#0MS;
   VMaster.Virtual.TON_TimeoutMovement.IN := FALSE;
   VMaster.Virtual.TON_Enable.PT := T#0MS;
   VMaster.Virtual.TON_Enable.IN := FALSE;
   VMasterBooked.PLS.Pos0.LowLimit := 5000.0;
   VMasterBooked.PLS.Pos0.HighLimit := 0.0;
   VMasterBooked.PLS.Pos0.Ok := FALSE;
   VMasterBooked.PLS.Pos1.LowLimit := 320.0;
   VMasterBooked.PLS.Pos1.HighLimit := 400.0;
   VMasterBooked.PLS.Pos1.Ok := FALSE;
   VMasterBooked.PLS.Pos2.LowLimit := 680.0;
   VMasterBooked.PLS.Pos2.HighLimit := 760.0;
   VMasterBooked.PLS.Pos2.Ok := FALSE;
   VMasterBooked.PLS.Pos3.LowLimit := 1040.0;
   VMasterBooked.PLS.Pos3.HighLimit := 1120.0;
   VMasterBooked.PLS.Pos3.Ok := FALSE;
   VMasterBooked.PLS.Pos4.LowLimit := 1400.0;
   VMasterBooked.PLS.Pos4.HighLimit := 1480.0;
   VMasterBooked.PLS.Pos4.Ok := FALSE;
   VMasterBooked.PLS.Pos5.LowLimit := 1760.0;
   VMasterBooked.PLS.Pos5.HighLimit := 1840.0;
   VMasterBooked.PLS.Pos5.Ok := FALSE;
   VMasterBooked.PLS.Pos6.LowLimit := 2120.0;
   VMasterBooked.PLS.Pos6.HighLimit := 2200.0;
   VMasterBooked.PLS.Pos6.Ok := FALSE;
   VMasterBooked.PLS.Pos7.LowLimit := 2480.0;
   VMasterBooked.PLS.Pos7.HighLimit := 2560.0;
   VMasterBooked.PLS.Pos7.Ok := FALSE;
   VMasterBooked.PLS.Pos8.LowLimit := 2840.0;
   VMasterBooked.PLS.Pos8.HighLimit := 2920.0;
   VMasterBooked.PLS.Pos8.Ok := FALSE;
   VMasterBooked.PLS.Pos9.LowLimit := 3200.0;
   VMasterBooked.PLS.Pos9.HighLimit := 3280.0;
   VMasterBooked.PLS.Pos9.Ok := FALSE;
   VMasterBooked.PLS.Pos10.LowLimit := 3560.0;
   VMasterBooked.PLS.Pos10.HighLimit := 3640.0;
   VMasterBooked.PLS.Pos10.Ok := FALSE;
   VMasterBooked.PLS.Pos11.LowLimit := 3920.0;
   VMasterBooked.PLS.Pos11.HighLimit := 4000.0;
   VMasterBooked.PLS.Pos11.Ok := FALSE;
   VMasterBooked.PLS.Pos12.LowLimit := 4280.0;
   VMasterBooked.PLS.Pos12.HighLimit := 4360.0;
   VMasterBooked.PLS.Pos12.Ok := FALSE;
   VMasterBooked.PLS.Pos13.LowLimit := 4640.0;
   VMasterBooked.PLS.Pos13.HighLimit := 4720.0;
   VMasterBooked.PLS.Pos13.Ok := FALSE;
   VMasterBooked.PLS.Pos14.LowLimit := 5000.0;
   VMasterBooked.PLS.Pos14.HighLimit := 5080.0;
   VMasterBooked.PLS.Pos14.Ok := FALSE;
   VMasterBooked.PLS.Pos15.LowLimit := 5360.0;
   VMasterBooked.PLS.Pos15.HighLimit := 5440.0;
   VMasterBooked.PLS.Pos15.Ok := FALSE;
   VMasterBooked.PLS.Pos16.LowLimit := 0.0;
   VMasterBooked.PLS.Pos16.HighLimit := 0.0;
   VMasterBooked.PLS.Pos16.Ok := FALSE;
   VMasterBooked.PLS.Pos17.LowLimit := 0.0;
   VMasterBooked.PLS.Pos17.HighLimit := 0.0;
   VMasterBooked.PLS.Pos17.Ok := FALSE;
   VMasterBooked.PLS.Pos18.LowLimit := 0.0;
   VMasterBooked.PLS.Pos18.HighLimit := 0.0;
   VMasterBooked.PLS.Pos18.Ok := FALSE;
   VMasterBooked.PLS.Pos19.LowLimit := 0.0;
   VMasterBooked.PLS.Pos19.HighLimit := 0.0;
   VMasterBooked.PLS.Pos19.Ok := FALSE;
   VMasterBooked.PLS.CM_CheckMouInf.LowLimit := 0.0;
   VMasterBooked.PLS.CM_CheckMouInf.HighLimit := 0.0;
   VMasterBooked.PLS.CM_CheckMouInf.Ok := FALSE;
   VMasterBooked.PLS.OM_CheckMouInf.LowLimit := 0.0;
   VMasterBooked.PLS.OM_CheckMouInf.HighLimit := 0.0;
   VMasterBooked.PLS.OM_CheckMouInf.Ok := FALSE;
   VMasterBooked.Man.EnaPbt := FALSE;
   VMasterBooked.Man.RstCmd := FALSE;
   VMasterBooked.Man.ScreenNumber := 300_100_301;
   VMasterBooked.Man.WithinScreenRange := 0;
   VMasterBooked.Virtual.AlmOk := TRUE;
   VMasterBooked.Virtual.AlmEmerg := FALSE;
   VMasterBooked.Virtual.AlmNode := FALSE;
   VMasterBooked.Virtual.InitPosDrive := TRUE;
   VMasterBooked.Virtual.InitPosDrivePLS := FALSE;
   VMasterBooked.Virtual.GearingON := TRUE;
   VMasterBooked.Virtual.CamHook := FALSE;
   VMasterBooked.Virtual.CamStoppingPhase := FALSE;
   VMasterBooked.Virtual.RepositioningRequest := FALSE;
   VMasterBooked.Virtual.CamRequestResult := FALSE;
   VMasterBooked.Virtual.CamRequestError := FALSE;
   VMasterBooked.Virtual.CamRequestOk := FALSE;
   VMasterBooked.Virtual.AuxCamRequest := FALSE;
   VMasterBooked.Virtual.Cmd_Repos := FALSE;
   VMasterBooked.Virtual.Ons_RedefinePosition := FALSE;
   VMasterBooked.Virtual.Ons_CamRequest := FALSE;
   VMasterBooked.Virtual.AuxCmdPosition := 0;
   VMasterBooked.Virtual.Cfg_FBK_In_Position_Delay_ms := 100;
   VMasterBooked.Virtual.Unwind := 5040.0;
   VMasterBooked.Virtual.MaxDev := 0.0;
   VMasterBooked.Virtual.ReposSpeed := 0.0;
   VMasterBooked.Virtual.CalcSlaveDifferenceABS := 0.0;
   VMasterBooked.Virtual.CalcModPosition := 0.0;
   VMasterBooked.Virtual.CalcSlaveDifference := 0.0;
   VMasterBooked.Virtual.CalcMinDeltaPos := 0.0;
   VMasterBooked.Virtual.CalcMaxDeltaPos := 0.0;
   VMasterBooked.Virtual.CalcHalfPosUnwind := 0.0;
   VMasterBooked.Virtual.Man.Cmd_PosJog := FALSE;
   VMasterBooked.Virtual.Man.Cmd_NegJog := FALSE;
   VMasterBooked.Virtual.Man.Cmd_Step := FALSE;
   VMasterBooked.Virtual.Man.Cmd_Forward := FALSE;
   VMasterBooked.Virtual.Man.Cmd_Backward := FALSE;
   VMasterBooked.Virtual.Man.Cmd_Up := FALSE;
   VMasterBooked.Virtual.Man.Cmd_Down := FALSE;
   VMasterBooked.Virtual.Man.Cmd_Intermediate := FALSE;
   VMasterBooked.Virtual.Man.Cmd_Open := FALSE;
   VMasterBooked.Virtual.Man.Cmd_Close := FALSE;
   VMasterBooked.Virtual.Man.Cmd_PreOpen := FALSE;
   VMasterBooked.Virtual.Man.Cmd_Maintenance := FALSE;
   VMasterBooked.Virtual.Man.Cmd_OperatorSide := FALSE;
   VMasterBooked.Virtual.Man.Cmd_NotOperatorSide := FALSE;
   VMasterBooked.Virtual.Man.Cmd_OnMould := FALSE;
   VMasterBooked.Virtual.Man.Cmd_OffMould := FALSE;
   VMasterBooked.Virtual.Man.Cmd_Pos0 := FALSE;
   VMasterBooked.Virtual.Man.Cmd_Pos1 := FALSE;
   VMasterBooked.Virtual.Man.Cmd_Pos2 := FALSE;
   VMasterBooked.Virtual.Man.Cmd_Pos3 := FALSE;
   VMasterBooked.Virtual.Man.Cmd_Pos4 := FALSE;
   VMasterBooked.Virtual.Man.Cmd_Pos5 := FALSE;
   VMasterBooked.Virtual.Man.Ons_Step := FALSE;
   VMasterBooked.Virtual.Man.PhaseJogCmd := FALSE;
   VMasterBooked.Virtual.Man.CmdStartStep := FALSE;
   VMasterBooked.Virtual.Man.CmdEndStep := FALSE;
   VMasterBooked.Virtual.Man.StepCond := FALSE;
   VMasterBooked.Virtual.Man.TON_DelayHomeCmd.PT := T#3S;
   VMasterBooked.Virtual.Man.TON_DelayHomeCmd.IN := FALSE;
   VMasterBooked.Virtual.Auto.Cmd_Step := FALSE;
   VMasterBooked.Virtual.Auto.Cmd_StartStep := FALSE;
   VMasterBooked.Virtual.Auto.Cmd_EndStep := FALSE;
   VMasterBooked.Virtual.Auto.Cmd_Forward := FALSE;
   VMasterBooked.Virtual.Auto.Cmd_Backward := FALSE;
   VMasterBooked.Virtual.Auto.Cmd_Up := FALSE;
   VMasterBooked.Virtual.Auto.Cmd_Down := FALSE;
   VMasterBooked.Virtual.Auto.Cmd_Intermediate := FALSE;
   VMasterBooked.Virtual.Auto.Cmd_Open := FALSE;
   VMasterBooked.Virtual.Auto.Cmd_Close := FALSE;
   VMasterBooked.Virtual.Auto.Cmd_PreOpen := FALSE;
   VMasterBooked.Virtual.Auto.Cmd_Maintenance := FALSE;
   VMasterBooked.Virtual.Auto.Cmd_OperatorSide := FALSE;
   VMasterBooked.Virtual.Auto.Cmd_NotOperatorSide := FALSE;
   VMasterBooked.Virtual.Auto.Cmd_OnMould := FALSE;
   VMasterBooked.Virtual.Auto.Cmd_OffMould := FALSE;
   VMasterBooked.Virtual.Auto.Cmd_Pos0 := FALSE;
   VMasterBooked.Virtual.Auto.Cmd_Pos1 := FALSE;
   VMasterBooked.Virtual.Auto.Cmd_Pos2 := FALSE;
   VMasterBooked.Virtual.Auto.Cmd_Pos3 := FALSE;
   VMasterBooked.Virtual.Auto.Cmd_Pos4 := FALSE;
   VMasterBooked.Virtual.Auto.Cmd_Pos5 := FALSE;
   VMasterBooked.Virtual.Auto.Cmd_Gear := FALSE;
   VMasterBooked.Virtual.ACT.CMD.Enable := TRUE;
   VMasterBooked.Virtual.ACT.CMD.Pos_Mode := FALSE;
   VMasterBooked.Virtual.ACT.CMD.MergeDisabled := FALSE;
   VMasterBooked.Virtual.ACT.CMD.SCurve := FALSE;
   VMasterBooked.Virtual.ACT.CMD.Cam_Mode := FALSE;
   VMasterBooked.Virtual.ACT.CMD.Cam_Request := FALSE;
   VMasterBooked.Virtual.ACT.CMD.Cam_PhaseStop := FALSE;
   VMasterBooked.Virtual.ACT.CMD.Gear_Mode := TRUE;
   VMasterBooked.Virtual.ACT.CMD.Repos_Req := FALSE;
   VMasterBooked.Virtual.ACT.CMD.Jog_Pos := FALSE;
   VMasterBooked.Virtual.ACT.CMD.Jog_Neg := FALSE;
   VMasterBooked.Virtual.ACT.CMD.Stop := FALSE;
   VMasterBooked.Virtual.ACT.CMD.Stop_InPhase := FALSE;
   VMasterBooked.Virtual.ACT.CMD.Stop_Emergency := FALSE;
   VMasterBooked.Virtual.ACT.CMD.Stop_Immediate := FALSE;
   VMasterBooked.Virtual.ACT.CMD.RedefinePosition := FALSE;
   VMasterBooked.Virtual.ACT.CMD.Calibration_Req := FALSE;
   VMasterBooked.Virtual.ACT.CMD.Reset := FALSE;
   VMasterBooked.Virtual.ACT.CMD.OneShootMove := FALSE;
   VMasterBooked.Virtual.ACT.CMD.SetPositionUnwind := FALSE;
   VMasterBooked.Virtual.ACT.CMD.Move_Type := 0;
   VMasterBooked.Virtual.ACT.CMD.Target_Pos := 0.0;
   VMasterBooked.Virtual.ACT.CMD.Speed := 0.0;
   VMasterBooked.Virtual.ACT.CMD.Acceleration := 0.0;
   VMasterBooked.Virtual.ACT.CMD.Deceleration := 750.0;
   VMasterBooked.Virtual.ACT.CMD.PositionUnwind := 0;
   VMasterBooked.Virtual.ACT.CMD.Mrp_Position := 558.0;
   VMasterBooked.Virtual.ACT.CMD.Gear_Ratio := 1.0;
   VMasterBooked.Virtual.ACT.CMD.Mccp_Length := 0;
   VMasterBooked.Virtual.ACT.CMD.Mccp_StartSlope := 0.0;
   VMasterBooked.Virtual.ACT.CMD.Mccp_EndSlope := 0.0;
   VMasterBooked.Virtual.ACT.CMD.Mapc_Direction := 0;
   VMasterBooked.Virtual.ACT.CMD.Mapc_SlaveScaling := 0.0;
   VMasterBooked.Virtual.ACT.CMD.Mapc_MasterScaling := 0.0;
   VMasterBooked.Virtual.ACT.CMD.Mapc_MasterLockPosition := 0.0;
   VMasterBooked.Virtual.ACT.CMD.Mapc_CamLockPosition := 0.0;
   VMasterBooked.Virtual.ACT.CMD.Cam[0..39].leadingValueStart := 0.0;
   VMasterBooked.Virtual.ACT.CMD.Cam[0..39].leadingValueEnd := 0.0;
   VMasterBooked.Virtual.ACT.CMD.Cam[0..39].followingValueStart := 0.0;
   VMasterBooked.Virtual.ACT.CMD.Cam[0..39].followingValueEnd := 0.0;
   VMasterBooked.Virtual.ACT.CMD.Cam[0..39].geoVeloStart := 0.0;
   VMasterBooked.Virtual.ACT.CMD.Cam[0..39].geoVeloEnd := 0.0;
   VMasterBooked.Virtual.ACT.CMD.Cam[0..39].geoAccelStart := 0.0;
   VMasterBooked.Virtual.ACT.CMD.Cam[0..39].geoAccelEnd := 0.0;
   VMasterBooked.Virtual.ACT.CMD.Cam[0..39].geoJerkStart := 0.0;
   VMasterBooked.Virtual.ACT.CMD.Cam[0..39].geoJerkEnd := 0.0;
   VMasterBooked.Virtual.ACT.CMD.Cam[0..39].inflectionPointParameter := 0.5;
   VMasterBooked.Virtual.ACT.CMD.Cam[0..39].modVeloTrapezoidParameter := 1.0;
   VMasterBooked.Virtual.ACT.CMD.Cam[0..39].modSineMaxAccelCaStar := 0.0;
   VMasterBooked.Virtual.ACT.CMD.Cam[0..39].camProfileType := 0;
   VMasterBooked.Virtual.ACT.FBK.Ready := TRUE;
   VMasterBooked.Virtual.ACT.FBK.Calibrated := TRUE;
   VMasterBooked.Virtual.ACT.FBK.MRP_DN := FALSE;
   VMasterBooked.Virtual.ACT.FBK.Fault := FALSE;
   VMasterBooked.Virtual.ACT.FBK.In_Position := TRUE;
   VMasterBooked.Virtual.ACT.FBK.Standstill := TRUE;
   VMasterBooked.Virtual.ACT.FBK.Enabled := TRUE;
   VMasterBooked.Virtual.ACT.FBK.Gearing_IP := TRUE;
   VMasterBooked.Virtual.ACT.FBK.Position := 655.68;
   VMasterBooked.Virtual.ACT.FBK.Speed := 0.0;
   VMasterBooked.Virtual.ACT.FBK.PositionUnwind := 0;
   VMasterBooked.Virtual.ACT.FBK.SeqCamErrorCode := 0;
   VMasterBooked.Virtual.ACT.FBK.SeqCamTargetPosMAM := 0.0;
   VMasterBooked.Virtual.ACT.FBK.SeqCamStatus.EndSequence := FALSE;
   VMasterBooked.Virtual.ACT.FBK.SeqCamStatus.EndSuccess := FALSE;
   VMasterBooked.Virtual.ACT.FBK.SeqCamStatus.EndError := FALSE;
   VMasterBooked.Virtual.ACT.FBK.SeqCamStatus.CamHook := FALSE;
   VMasterBooked.Virtual.ACT.FBK.SeqCamStatus.BothMapc_IP := FALSE;
   VMasterBooked.Virtual.ACT.FBK.SeqCamStatus.SlaveFwd := FALSE;
   VMasterBooked.Virtual.ACT.FBK.SeqCamStatus.SlaveBwd := FALSE;
   VMasterBooked.Virtual.ACT.FBK.SeqCamStatus.SlaveUnwind := FALSE;
   VMasterBooked.Virtual.ACT.FBK.SeqCamStatus.WaitValidByOpe := FALSE;
   VMasterBooked.Virtual.ACT.FBK.SeqCamStatus.MapcA_IP := FALSE;
   VMasterBooked.Virtual.ACT.FBK.SeqCamStatus.MapcB_IP := FALSE;
   VMasterBooked.Virtual.ACT.FBK.SeqCamStatus.MapcC_IP := FALSE;
   VMasterBooked.Virtual.ACT.FBK.SeqCamStatus.CamOnce_PC := FALSE;
   VMasterBooked.Virtual.ACT.FBK.SeqCamStatus.MaxDevError := FALSE;
   VMasterBooked.Virtual.ACT.FBK.SeqCamStatus.PositionCamLockStatus := FALSE;
   VMasterBooked.Virtual.ACT.FBK.SeqCamStatus.WaitRestart := FALSE;
   VMasterBooked.Virtual.ACT.FBK.SeqCamStatus.Bit17 := FALSE;
   VMasterBooked.Virtual.ACT.FBK.SeqCamStatus.Bit18 := FALSE;
   VMasterBooked.Virtual.ACT.FBK.SeqCamStatus.Bit19 := FALSE;
   VMasterBooked.Virtual.ACT.FBK.SeqCamStatus.Bit20 := FALSE;
   VMasterBooked.Virtual.ACT.FBK.SeqCamStatus.Bit21 := FALSE;
   VMasterBooked.Virtual.ACT.FBK.SeqCamStatus.Bit22 := FALSE;
   VMasterBooked.Virtual.ACT.FBK.SeqCamStatus.Bit23 := FALSE;
   VMasterBooked.Virtual.ACT.FBK.SeqCamStatus.Bit24 := FALSE;
   VMasterBooked.Virtual.ACT.FBK.SeqCamStatus.Bit25 := FALSE;
   VMasterBooked.Virtual.ACT.FBK.SeqCamStatus.Bit26 := FALSE;
   VMasterBooked.Virtual.ACT.FBK.SeqCamStatus.Bit27 := FALSE;
   VMasterBooked.Virtual.ACT.FBK.SeqCamStatus.Bit28 := FALSE;
   VMasterBooked.Virtual.ACT.FBK.SeqCamStatus.Bit29 := FALSE;
   VMasterBooked.Virtual.ACT.FBK.SeqCamStatus.Bit30 := FALSE;
   VMasterBooked.Virtual.ACT.FBK.SeqCamStatus.Bit31 := FALSE;
   VMasterBooked.Virtual.ACT.FBK.SeqCamStatus.Bit32 := FALSE;
   VMasterBooked.Virtual.PLS.FinePosOk.LowLimit := 0.0;
   VMasterBooked.Virtual.PLS.FinePosOk.HighLimit := 0.0;
   VMasterBooked.Virtual.PLS.FinePosOk.Ok := FALSE;
   VMasterBooked.Virtual.PLS.KeepPosOk.LowLimit := 0.0;
   VMasterBooked.Virtual.PLS.KeepPosOk.HighLimit := 0.0;
   VMasterBooked.Virtual.PLS.KeepPosOk.Ok := FALSE;
   VMasterBooked.Virtual.PLS.Up.LowLimit := 0.0;
   VMasterBooked.Virtual.PLS.Up.HighLimit := 0.0;
   VMasterBooked.Virtual.PLS.Up.Ok := FALSE;
   VMasterBooked.Virtual.PLS.Intermediate.LowLimit := 0.0;
   VMasterBooked.Virtual.PLS.Intermediate.HighLimit := 0.0;
   VMasterBooked.Virtual.PLS.Intermediate.Ok := FALSE;
   VMasterBooked.Virtual.PLS.Down.LowLimit := 0.0;
   VMasterBooked.Virtual.PLS.Down.HighLimit := 0.0;
   VMasterBooked.Virtual.PLS.Down.Ok := FALSE;
   VMasterBooked.Virtual.PLS.Forward.LowLimit := 0.0;
   VMasterBooked.Virtual.PLS.Forward.HighLimit := 0.0;
   VMasterBooked.Virtual.PLS.Forward.Ok := FALSE;
   VMasterBooked.Virtual.PLS.Backward.LowLimit := 0.0;
   VMasterBooked.Virtual.PLS.Backward.HighLimit := 0.0;
   VMasterBooked.Virtual.PLS.Backward.Ok := FALSE;
   VMasterBooked.Virtual.PLS.Open.LowLimit := 0.0;
   VMasterBooked.Virtual.PLS.Open.HighLimit := 0.0;
   VMasterBooked.Virtual.PLS.Open.Ok := FALSE;
   VMasterBooked.Virtual.PLS.Close.LowLimit := 0.0;
   VMasterBooked.Virtual.PLS.Close.HighLimit := 0.0;
   VMasterBooked.Virtual.PLS.Close.Ok := FALSE;
   VMasterBooked.Virtual.PLS.PreOpen.LowLimit := 0.0;
   VMasterBooked.Virtual.PLS.PreOpen.HighLimit := 0.0;
   VMasterBooked.Virtual.PLS.PreOpen.Ok := FALSE;
   VMasterBooked.Virtual.PLS.Maintenance.LowLimit := 0.0;
   VMasterBooked.Virtual.PLS.Maintenance.HighLimit := 0.0;
   VMasterBooked.Virtual.PLS.Maintenance.Ok := FALSE;
   VMasterBooked.Virtual.PLS.OperatorSide.LowLimit := 0.0;
   VMasterBooked.Virtual.PLS.OperatorSide.HighLimit := 0.0;
   VMasterBooked.Virtual.PLS.OperatorSide.Ok := FALSE;
   VMasterBooked.Virtual.PLS.NotOperatorSide.LowLimit := 0.0;
   VMasterBooked.Virtual.PLS.NotOperatorSide.HighLimit := 0.0;
   VMasterBooked.Virtual.PLS.NotOperatorSide.Ok := FALSE;
   VMasterBooked.Virtual.PLS.OnMould.LowLimit := 0.0;
   VMasterBooked.Virtual.PLS.OnMould.HighLimit := 0.0;
   VMasterBooked.Virtual.PLS.OnMould.Ok := FALSE;
   VMasterBooked.Virtual.PLS.OffMould.LowLimit := 0.0;
   VMasterBooked.Virtual.PLS.OffMould.HighLimit := 0.0;
   VMasterBooked.Virtual.PLS.OffMould.Ok := FALSE;
   VMasterBooked.Virtual.PLS.Pos0.LowLimit := 0.0;
   VMasterBooked.Virtual.PLS.Pos0.HighLimit := 0.0;
   VMasterBooked.Virtual.PLS.Pos0.Ok := FALSE;
   VMasterBooked.Virtual.PLS.Pos1.LowLimit := 0.0;
   VMasterBooked.Virtual.PLS.Pos1.HighLimit := 0.0;
   VMasterBooked.Virtual.PLS.Pos1.Ok := FALSE;
   VMasterBooked.Virtual.PLS.Pos2.LowLimit := 0.0;
   VMasterBooked.Virtual.PLS.Pos2.HighLimit := 0.0;
   VMasterBooked.Virtual.PLS.Pos2.Ok := FALSE;
   VMasterBooked.Virtual.PLS.Pos3.LowLimit := 0.0;
   VMasterBooked.Virtual.PLS.Pos3.HighLimit := 0.0;
   VMasterBooked.Virtual.PLS.Pos3.Ok := FALSE;
   VMasterBooked.Virtual.PLS.Pos4.LowLimit := 0.0;
   VMasterBooked.Virtual.PLS.Pos4.HighLimit := 0.0;
   VMasterBooked.Virtual.PLS.Pos4.Ok := FALSE;
   VMasterBooked.Virtual.PLS.Pos5.LowLimit := 0.0;
   VMasterBooked.Virtual.PLS.Pos5.HighLimit := 0.0;
   VMasterBooked.Virtual.PLS.Pos5.Ok := FALSE;
   VMasterBooked.Virtual.TON_TimeoutMovement.PT := T#0MS;
   VMasterBooked.Virtual.TON_TimeoutMovement.IN := FALSE;
   VMasterBooked.Virtual.TON_Enable.PT := T#0MS;
   VMasterBooked.Virtual.TON_Enable.IN := FALSE;
END_DATA_BLOCK
